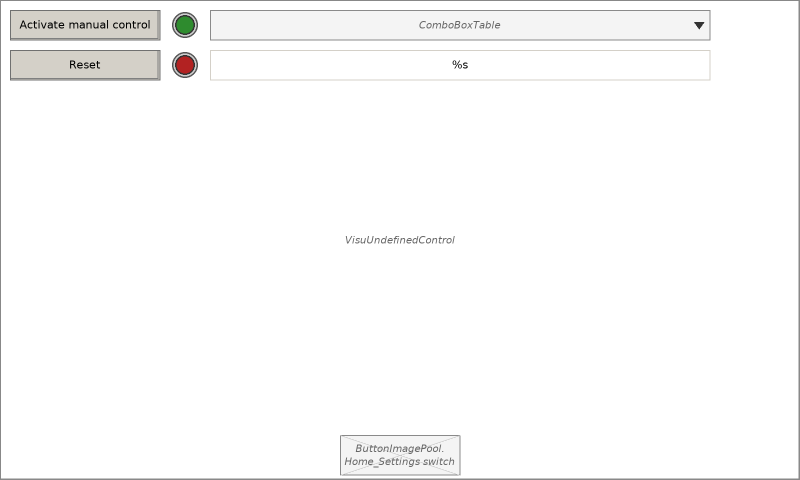
VISUALIZATION ManualControl  // 800x480
    Frame (0,0 800x480), input disabled if: GVL_DevManual.fbManualControler.bDisableManualInputs, frame switch variable: GVL_DevManual.fbManualControler.eDevType
        shows VisuUndefinedControl()
        shows VisuValveControl()
        shows VisuCylinderControl()
        shows VisuAxisControl()
        shows VisuPushbuttonLightControl()
        shows VisuDigitalInputControl()
        shows VisuAnlogInputControl()
        shows VisuDigitalOutControl()
        shows VisuAnalogOutControl()
        shows VisuPWMControl()
        shows VisuDoublePWMControl()
    Button (10,10 150x30), "Activate manual control", pressed state: GVL_DevManual.fbManualControler.bManualActive
        toggle GVL_DevManual.fbManualControler.bManualActive
    Lamp1 (170,50 30x30), tooltip "component fault active", variable: GVL_DevManual.fbManualControler.bErroractive, style: Lamp-Lamp1-Red
    Lamp1 (170,10 30x30), tooltip "Manual control active", variable: GVL_DevManual.fbManualControler.bManual, style: Lamp-Lamp1-Green
    Textfield (210,50 500x30), "%s", text variable: GVL_DevManual.fbManualControler.sDeviceState
    Button (10,50 150x30), "Reset"
        tap GVL_DevManual.fbManualControler.bReset
    ComboBoxTable (210,10 500x30), variable: GVL_DevManual.fbManualControler.nCmdLookupindex, data array: GVL_DevManual.fbManualControler.arDeviceArray
        p3854506369: GVL_DevManual.fbManualControler.arDeviceArray[INDEX].sName
        p1892666644: GVL_DevManual.fbManualControler.arDeviceArray[INDEX].sType
        p338671338: GVL_DevManual.fbManualControler.arDeviceArray[INDEX].pFunction^
        p1128707560: GVL_DevManual.fbManualControler.nNumberOfDevices
    Image (340,435 120x40), image: ButtonImagePool.Home_Settings switch
        OnMouseClick: execute { GVL_HMI.nStartVisu := E_StartVisu.Logo ; }
        OnMouseClick: toggle GVL_Parameters.fbParameterHandler.bCmdParFileWrite
END_VISUALIZATION

(* stored: Version 1.1.0.1, ProductVersion 3.1.4024.5
   Visu ManualControl: Id {47fd7eab-4722-4161-bb7e-85fd17bf2676} *)
